// abstracts the ARCommunicationWSExtention
FUNCTION_BLOCK ARCommunicationWS_t 
VAR_INPUT
END_VAR
VAR_OUTPUT
END_VAR
VAR
	_ARDevice : ARCommunicationWSExtentionWS_t;
	_initialConnect : BOOL := FALSE;
END_VAR

METHOD getConnectionStatus : BOOL
VAR_INPUT
END_VAR
// gets the communication status of the connection
getConnectionStatus := _ARDevice.bConnected;
return;
END_METHOD

// gets the last saved message from the client (max str length 255)
METHOD getLastMessage : STRING(255)
VAR_INPUT
END_VAR
getLastMessage := _ARDevice.lastMessage;

_ARDevice.newMessageAvalable := FALSE;
END_METHOD

METHOD newMessageRecived : BOOL
VAR_INPUT
END_VAR
// returns if a new message has been recived
newMessageRecived := _ARDevice._newMessageAvalable;
END_METHOD

METHOD sendNewMessage : BOOL
VAR_INPUT
	str : STRING(255); // (max str length 255)
END_VAR
// sends a new message to the client
_ARDevice.SendMessage(pContent := ADR(str), nContentSize := SIZEOF(str), bTextContent := TRUE, bCompress := FALSE);
END_METHOD

METHOD PRIVATE startConnection : BOOL
VAR_INPUT
END_VAR
IF _ARDevice.bConnected THEN
	RETURN;
END_IF


_ARDevice.nHostPort := 1880;
_ARDevice.sHostName := 'localhost';
_ARDevice.sUri := 'ws/PLC';
_ARDevice.bKeepAlive := FALSE;
_ARDevice.nConnectResponseTimeout := 60;
_ARDevice.nKeepAliveCloseTimeout := 60;
//_ARDevice.stTLS.bNoServerCertCheck := TRUE;
_ARDevice.bPerMessageDeflate := FALSE;
_ARDevice.sOrigin := 'ws/PLC';
_ARDevice.Connect(TRUE);
END_METHOD

METHOD PRIVATE stopConnection : BOOL
VAR_INPUT
END_VAR
IF NOT _ARDevice.bConnected THEN
	RETURN;
END_IF

_ARDevice.Disconnect();
END_METHOD

// is called every cycle, used to upholed communication and check if a new message has been recived
METHOD update : BOOL
VAR_INPUT
END_VAR
IF _initialConnect = FALSE THEN // initial connection
	_initialConnect := true;
	THIS^.startConnection();
END_IF

IF _ARDevice.eConnectionState = ETcIotWebSocketStatus.WS_STATUS_SOCK_NO_CONN THEN 
	//THIS^.stopConnection();
END_IF

IF _ARDevice.bConnected = FALSE AND _ARDevice.eConnectionState <> ETcIotWebSocketStatus.WS_STATUS_BUSY THEN // retry if connection is lost
	//THIS^.startConnection();
END_IF

_ARDevice.Execute();
END_METHOD

END_FUNCTION_BLOCK

(* stored: Version 1.1.0.1
   POU ARCommunicationWS_t: Id {3697f1d2-5144-45fb-a78b-bb7912cd4429}, SpecialFunc None
   Method getConnectionStatus: Id {e629fbae-7329-41fc-8f52-af6f3d5840fa}
   Method getLastMessage: Id {08a227d9-9e52-499f-99b3-521fa34ba409}
   Method newMessageRecived: Id {ebfdd1a5-1abb-4bc2-b017-ad4dd8dc6e08}
   Method sendNewMessage: Id {7ab18af5-7bc5-4c96-b223-14eb6cce1ab3}
   Method startConnection: Id {89d039a8-3323-4f6e-9842-93aae51be57a}
   Method stopConnection: Id {95fcb138-8ce0-4fcb-8c62-1a615f795ab1}
   Method update: Id {25efbe41-3ef8-45cc-91e3-4ad477496cc8} *)
